TYPE St_Assy_SignOff EXTENDS St_Assy_Base :
STRUCT
END_STRUCT
END_TYPE

(* stored: Version 1.1.0.1
   DUT St_Assy_SignOff: Id {78985a90-5378-4de3-a390-b2f8b589fae9} *)
